TYPE ZData :
STRUCT
  Config : ZDataConfig;
  Machine : ZDataMachine;
  Calibration : ZDataCalibration;
  Recipe : ZDataRecipe;
END_STRUCT
END_TYPE

(* stored: Version 1.1.0.1
   DUT ZData: Id {073363c1-2230-4d70-a034-086af5048cff} *)
